% RSLogix 500 project ESTACION1.RSS, saved by version 8.40.00.08 %
PROJECT "UNTITLED"    % processor: MicroLogix 1500 %

PROGRAM FILES
  LAD 2   7 rungs

DATA FILES
  O0 OUTPUT  4 elements
  I1 INPUT  4 elements
  S2 STATUS  66 elements
  B3 BINARY  1 elements
  T4 TIMER  2 elements
  C5 COUNTER  1 elements
  R6 CONTROL  1 elements
  N7 INTEGER  1 elements
  F8 FLOAT  1 elements

LADDER 2
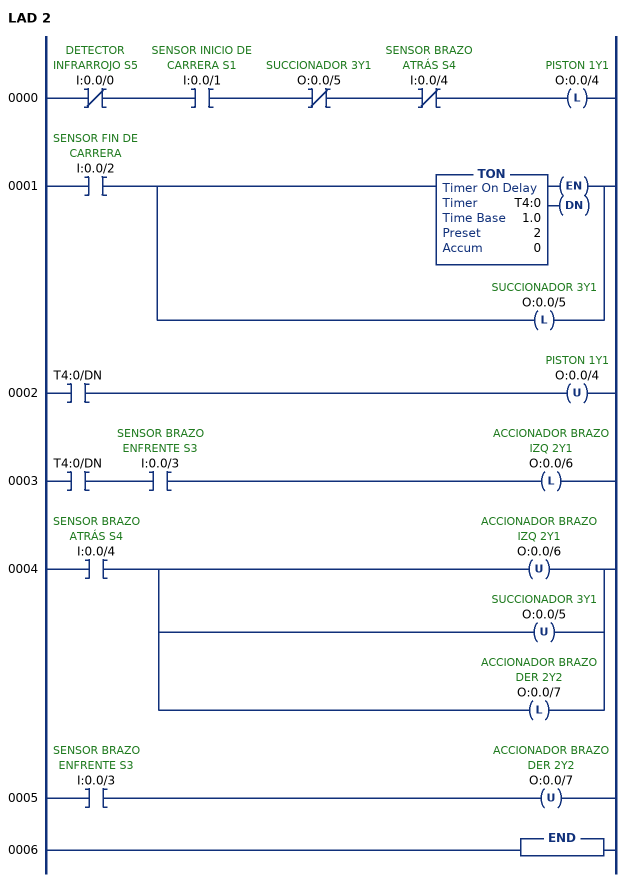
% Rung: 0 %
SOR XIO I:0.0/0 XIC I:0.0/1 XIO O:0.0/5 XIO I:0.0/4 OTL O:0.0/4 EOR
%   I:0.0/0  "DETECTOR INFRARROJO S5" %
%   I:0.0/1  "SENSOR INICIO DE CARRERA S1" %
%   O:0.0/5  "SUCCIONADOR 3Y1" %
%   I:0.0/4  "SENSOR BRAZO ATRÁS S4" %
%   O:0.0/4  "PISTON 1Y1" %
% Rung: 1 %
SOR XIC I:0.0/2 BST TON T4:0 1.0 2 0 NXB OTL O:0.0/5 BND EOR
%   I:0.0/2  "SENSOR FIN DE CARRERA" %
%   O:0.0/5  "SUCCIONADOR 3Y1" %
% Rung: 2 %
SOR XIC T4:0/DN OTU O:0.0/4 EOR
%   O:0.0/4  "PISTON 1Y1" %
% Rung: 3 %
SOR XIC T4:0/DN XIC I:0.0/3 OTL O:0.0/6 EOR
%   I:0.0/3  "SENSOR BRAZO ENFRENTE S3" %
%   O:0.0/6  "ACCIONADOR BRAZO IZQ 2Y1" %
% Rung: 4 %
SOR XIC I:0.0/4 BST OTU O:0.0/6 NXB BST OTU O:0.0/5 NXB OTL O:0.0/7 BND BND EOR
%   I:0.0/4  "SENSOR BRAZO ATRÁS S4" %
%   O:0.0/6  "ACCIONADOR BRAZO IZQ 2Y1" %
%   O:0.0/5  "SUCCIONADOR 3Y1" %
%   O:0.0/7  "ACCIONADOR BRAZO DER 2Y2" %
% Rung: 5 %
SOR XIC I:0.0/3 OTU O:0.0/7 EOR
%   I:0.0/3  "SENSOR BRAZO ENFRENTE S3" %
%   O:0.0/7  "ACCIONADOR BRAZO DER 2Y2" %
% Rung: 6 %
SOR END EOR

OTHER DOCUMENTED ADDRESSES
  O:0.0/8  "ACCIONADOR BRAZO DER 2Y2"
  T4:1/DN  "ESPERA A QUE SUCCIONE LA PIEZA"

DATA TABLE (non-zero values as saved)
DATA T4
% .PRE .ACC %
% T4:0 % 2 0
% T4:1 % 2 0
